// Gets the lower bound index of the array of specified type.
FUNCTION F_GetInterfaceArrayLowerBound : T_Position // The lower bound index of the specified array.
VAR_IN_OUT
	arArray : ARRAY[*] OF __SYSTEM.IQueryInterface; // The array to query.
END_VAR

F_GetInterfaceArrayLowerBound := LOWER_BOUND(arArray, 1);

END_FUNCTION

(* stored: Version 1.1.0.1
   POU F_GetInterfaceArrayLowerBound: Id {3146c2fa-76c4-0127-1927-b73370a46120}, SpecialFunc None *)
